// TIA Portal V17 export
// export: Created 2025-01-08T13:55:36.7441231Z, ExportSetting WithDefaults, DisplayName Totally Integrated Automation Portal, DisplayVersion V17, DisplayName TIA Portal Openness, DisplayVersion V17, DisplayName TIA Portal Version Control Interface, DisplayVersion V17, DisplayName SINAMICS Startdrive Advanced, DisplayVersion V17 Update2, DisplayName SINAMICS Startdrive G130, G150, S120, S150, SINAMICS MV, S210, DisplayVersion V17 Update2, DisplayName SINAMICS Startdrive G110M, G120, G120C, G120D, G120P, G115D, DisplayVersion V17 Update2, DisplayName STEP 7 Professional, DisplayVersion V17, DisplayName STEP 7 Safety, DisplayVersion V17, DisplayName WinCC Advanced, DisplayVersion V17
TYPE "HSMConfigParaMask2"
// stored: IsFailsafeCompliant false
   STRUCT
      iSyncOutput3Delay : Bool;
      iSyncOutput3Lenght : Bool;
      iPreFeedLenght : Bool;
      iConveyorSpeed_1 : Bool;
      iConveyorSpeed_2 : Bool;
      iReserved_1 : Bool;
      iReserved_2 : Bool;
      iReserved_3 : Bool;
      iReserved_4 : Bool;
      iReserved_5 : Bool;
      iReserved_6 : Bool;
      iReserved_7 : Bool;
      iReserved_8 : Bool;
      iReserved_9 : Bool;
      iReserved_10 : Bool;
      iReserved_11 : Bool;
   END_STRUCT;
END_TYPE
